DATA_BLOCK DB 554
TITLE =
{ S7_techparam := 'S7WRTX.TCONT_CP' }
AUTHOR : SIMATIC
FAMILY : CONTROL
VERSION : 0.0

"TCONT_CP"
BEGIN
   PV_IN := 0.000000e+000;
   PV_PER := 0;
   DISV := 0.000000e+000;
   INT_HPOS := FALSE;
   INT_HNEG := FALSE;
   SELECT := 0;
   PV := 0.000000e+000;
   LMN := 0.000000e+000;
   LMN_PER := 0;
   QPULSE := FALSE;
   QLMN_HLM := FALSE;
   QLMN_LLM := FALSE;
   QC_ACT := TRUE;
   CYCLE := 1.000000e-001;
   CYCLE_P := 2.000000e-002;
   SP_INT := 0.000000e+000;
   MAN := 0.000000e+000;
   COM_RST := FALSE;
   MAN_ON := TRUE;
   DEADB_W := 0.000000e+000;
   I_ITLVAL := 0.000000e+000;
   LMN_HLM := 1.000000e+002;
   LMN_LLM := 0.000000e+000;
   PV_FAC := 1.000000e+000;
   PV_OFFS := 0.000000e+000;
   LMN_FAC := 1.000000e+000;
   LMN_OFFS := 0.000000e+000;
   PER_TM := 1.000000e+000;
   P_B_TM := 0.000000e+000;
   TUN_DLMN := 2.000000e+001;
   PER_MODE := 0;
   PVPER_ON := FALSE;
   I_ITL_ON := FALSE;
   PULSE_ON := FALSE;
   TUN_KEEP := FALSE;
   ER := 0.000000e+000;
   LMN_P := 0.000000e+000;
   LMN_I := 0.000000e+000;
   LMN_D := 0.000000e+000;
   PHASE := 0;
   STATUS_H := 0;
   STATUS_D := 0;
   QTUN_RUN := FALSE;
   PI_CON.GAIN := 0.000000e+000;
   PI_CON.TI := 0.000000e+000;
   PID_CON.GAIN := 0.000000e+000;
   PID_CON.TI := 0.000000e+000;
   PID_CON.TD := 0.000000e+000;
   PAR_SAVE.PFAC_SP := 1.000000e+000;
   PAR_SAVE.GAIN := 0.000000e+000;
   PAR_SAVE.TI := 0.000000e+000;
   PAR_SAVE.TD := 0.000000e+000;
   PAR_SAVE.D_F := 5.000000e+000;
   PAR_SAVE.CON_ZONE := 1.000000e+002;
   PAR_SAVE.CONZ_ON := FALSE;
   PFAC_SP := 1.000000e+000;
   GAIN := 2.000000e+000;
   TI := 4.000000e+001;
   TD := 1.000000e+001;
   D_F := 5.000000e+000;
   CON_ZONE := 1.000000e+002;
   CONZ_ON := FALSE;
   TUN_ON := FALSE;
   TUN_ST := FALSE;
   UNDO_PAR := FALSE;
   SAVE_PAR := FALSE;
   LOAD_PID := FALSE;
   PID_ON := TRUE;
   GAIN_P := 0.000000e+000;
   TU := 0.000000e+000;
   TA := 0.000000e+000;
   KIG := 0.000000e+000;
   N_PTN := 0.000000e+000;
   TM_LAG_P := 0.000000e+000;
   T_P_INF := 0.000000e+000;
   P_INF := 0.000000e+000;
   LMN0 := 0.000000e+000;
   PV0 := 0.000000e+000;
   PVDT0 := 0.000000e+000;
   PVDT := 0.000000e+000;
   PVDT_MAX := 0.000000e+000;
   NOI_PVDT := 0.000000e+000;
   NOISE_PV := 0.000000e+000;
   FIL_CYC := 1;
   POI_CMAX := 0;
   POI_CYCL := 0;
   sctFil := 0;
   srPv := 0.000000e+000;
   srNoise := 0.000000e+000;
   srPvdt2 := 0.000000e+000;
   srPvdtMax2 := 0.000000e+000;
   srNoise2 := 0.000000e+000;
   srPvOld2 := 0.000000e+000;
   siStatus := 0;
   siSpDir := 0;
   srTime := 0.000000e+000;
   sPvOld := 0.000000e+000;
   sSpOld := 0.000000e+000;
   srPvMin := 0.000000e+000;
   srPVsim := 0.000000e+000;
   srEffDlmn := 0.000000e+000;
   sInvAlt := 0.000000e+000;
   sIanteilAlt := 0.000000e+000;
   sRestInt := 0.000000e+000;
   sRestDif := 0.000000e+000;
   sRueck := 0.000000e+000;
   sLmn := 0.000000e+000;
   spassPTm := 0.000000e+000;
   sCycTmPass := 0.000000e+000;
   sPTm := 0.000000e+000;
   srOptLmn := 0.000000e+000;
   sbOptLmn := FALSE;
   sbConzOn := FALSE;
   sbSpChange := FALSE;
   sbReOpt := FALSE;
   sLmnHlmOld := 1.000000e+002;
   sLmnLlmOld := 0.000000e+000;
   srDiffSp := 0.000000e+000;
   siTime := L#0;
   siCycle := L#0;
   siCycleP := L#0;
   siPulsFil := 0;
   srPulsPv := 0.000000e+000;
   srDPvdt := 0.000000e+000;
   srDPvdt2 := 0.000000e+000;
   sNpInf := 0.000000e+000;
   sCycleM := 0.000000e+000;
   sGf11_30 := 0.000000e+000;
   sGf12_30 := 0.000000e+000;
   sGf21_30 := 0.000000e+000;
   sGf22_30 := 0.000000e+000;
   sPv0Sim_30 := 0.000000e+000;
   srPVsim3_30 := 0.000000e+000;
   srPVsim2_30 := 0.000000e+000;
   srPVsim1_30 := 0.000000e+000;
   srDelPvsim_30 := 0.000000e+000;
   sGf11_20 := 0.000000e+000;
   sGf12_20 := 0.000000e+000;
   sGf21_20 := 0.000000e+000;
   sGf22_20 := 0.000000e+000;
   sPv0Sim_20 := 0.000000e+000;
   srPVsim2_20 := 0.000000e+000;
   srPVsim1_20 := 0.000000e+000;
   srDelPvsim_20 := 0.000000e+000;
   sGf11_15 := 0.000000e+000;
   sGf12_15 := 0.000000e+000;
   sGf21_15 := 0.000000e+000;
   sGf22_15 := 0.000000e+000;
   sPv0Sim_15 := 0.000000e+000;
   srPVsim2_15 := 0.000000e+000;
   srPVsim1_15 := 0.000000e+000;
   srDelPvsim_15 := 0.000000e+000;
END_DATA_BLOCK

